// TIA Portal V20 export
TYPE "DT_DataToSafety"
// stored: IsFailsafeCompliant true
   STRUCT
      OpenShutterButton : Bool;
      ResetEmergencyStop : Bool;
      JOG_Mod : Bool;
      Activation_Axis : Bool;
      CloseShutter : Bool;
      FrontDoorLock : Bool;
      DoorsInhibit : Bool;
   END_STRUCT;
END_TYPE
